Omron Sysmac Studio project MQTT_example_project (Sysmac Studio 1.47.0.64008, StandardProject)

# Controller CPU0: NX1P2-9024DT1 version 1.46
Task PrimaryTask (priority 4, period or condition 2000): Program0
Library OmronLib_MQTT_Comm_V1_0 1.0.0 (contents left out)
Library JSONDecoding 0.0.9 (contents left out)
Library JSON 0.0.55 (contents left out)

VAR_GLOBAL
    connectionSettingsLocal : OmronLib\MQTT_Comm\sConnectionSettings;
    clientReference : OmronLib\MQTT_Comm\sClientReference;
    clientReferenceLocal : OmronLib\MQTT_Comm\sClientReference;
    JSON_BUFFER : JSON\JSONBuffer;
    JSON_STRING : STRING[1986];
END_VAR

PROGRAM Program0
VAR
    Pub_Topic : STRING[512];
    Pub_PubMsg : STRING[256];
    Pub_PubSettings : OmronLib\MQTT_Comm\sPubFlags;
    Sub_Topic : String[512];
    Connect : BOOL;
    i_FB_MQTTClient : OmronLib\MQTT_Comm\MQTTClient;
    ErrorPresent : BOOL;
    ErrorID : WORD;
    ErrorIDEx : DWORD;
    sendString : BOOL;
    i_FB_MQTTPubString : OmronLib\MQTT_Comm\MQTTPubString;
    Pub_PacketID : UINT;
    Pub_MsgType : USINT;
    i_FB_MQTTClientLocal : OmronLib\MQTT_Comm\MQTTClient;
    i_FB_Randomizer : Rand;
    randomizer : LREAL;
    temp_val : REAL;
END_VAR
VAR_EXTERNAL
    connectionSettingsLocal : OmronLib\MQTT_Comm\sConnectionSettings;
    clientReference : OmronLib\MQTT_Comm\sClientReference;
    clientReferenceLocal : OmronLib\MQTT_Comm\sClientReference;
    JSON_BUFFER : JSON\JSONBuffer;
    JSON_STRING : STRING[1986];
END_VAR

(* Section JSON_Formatting: ladder, written here as Structured Text *)

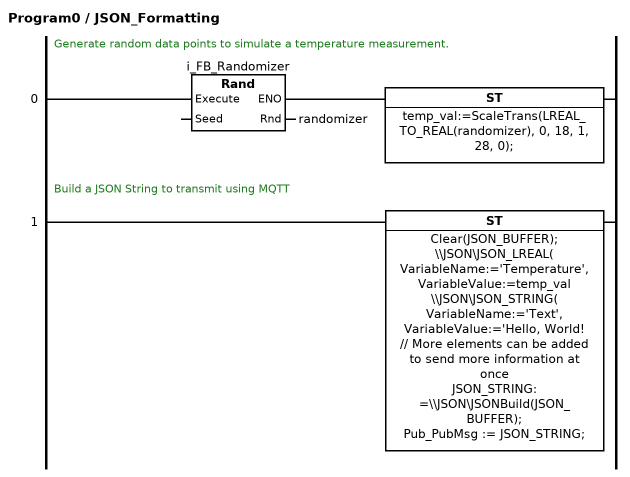
(* Rung 0: Generate random data points to simulate a temperature measurement. *)
i_FB_Randomizer(Execute := TRUE, Rnd => randomizer);
IF i_FB_Randomizer.ENO THEN
    temp_val:=ScaleTrans(LREAL_TO_REAL(randomizer), 0, 18, 1, 28, 0);
END_IF;
(* Rung 1: Build a JSON String to transmit using MQTT *)
Clear(JSON_BUFFER);																																		// Clear the JSON String buffer
\\JSON\JSON_LREAL(VariableName:='Temperature', VariableValue:=temp_val, Buffer:=JSON_BUFFER);		// Add first element to the JSON String
\\JSON\JSON_STRING(VariableName:='Text', VariableValue:='Hello, World!', Buffer:=JSON_BUFFER);			// Add second element to the JSON String

// More elements can be added to send more information at once

JSON_STRING:=\\JSON\JSONBuild(JSON_BUFFER);																						// Build a complete JSON String
Pub_PubMsg := JSON_STRING;

(* Section MQTT_Local: ladder, written here as Structured Text *)

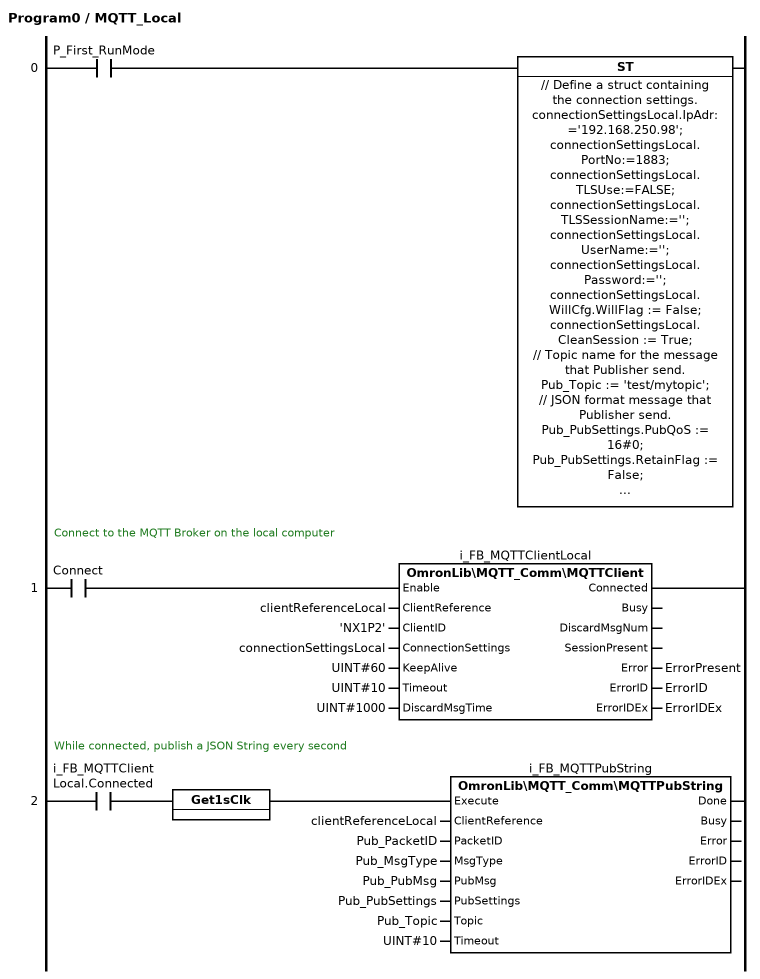
(* Rung 0 *)
IF P_First_RunMode THEN
    // Define a struct containing the connection settings. 
    connectionSettingsLocal.IpAdr:='192.168.250.98';
    connectionSettingsLocal.PortNo:=1883;
    connectionSettingsLocal.TLSUse:=FALSE;
    connectionSettingsLocal.TLSSessionName:='';
    connectionSettingsLocal.UserName:='';
    connectionSettingsLocal.Password:='';
    connectionSettingsLocal.WillCfg.WillFlag := False;
    connectionSettingsLocal.CleanSession := True;
    
    
    // Topic name for the message that Publisher send.
    Pub_Topic := 'test/mytopic';
    
    // JSON format message that Publisher send.
    Pub_PubSettings.PubQoS := 16#0;
    Pub_PubSettings.RetainFlag := False;
    
    // Topic name for the message that Subscriber receive.
    Sub_Topic := 'test/#';
END_IF;
(* Rung 1: Connect to the MQTT Broker on the local computer *)
i_FB_MQTTClientLocal(Enable := Connect, ClientReference := clientReferenceLocal, ClientID := 'NX1P2', ConnectionSettings := connectionSettingsLocal, KeepAlive := UINT#60, Timeout := UINT#10, DiscardMsgTime := UINT#1000, Error => ErrorPresent, ErrorID => ErrorID, ErrorIDEx => ErrorIDEx);
(* Rung 2: While connected, publish a JSON String every second *)
i_FB_MQTTPubString(Execute := i_FB_MQTTClientLocal.Connected AND Get1sClk(), ClientReference := clientReferenceLocal, PacketID := Pub_PacketID, MsgType := Pub_MsgType, PubMsg := Pub_PubMsg, PubSettings := Pub_PubSettings, Topic := Pub_Topic, Timeout := UINT#10);
END_PROGRAM